FUNCTION_BLOCK FB_FactoryIO_Lamp
VAR_INPUT
    bOn : BOOL;
END_VAR

VAR_OUTPUT
    OutSignal : BOOL;
END_VAR

OutSignal := bOn;

END_FUNCTION_BLOCK

(* stored: Version 1.1.0.1
   POU FB_FactoryIO_Lamp: Id {d0eaf3be-7893-4330-b027-41bd2241c42b}, SpecialFunc None *)
